Fanuc KAREL source: kt00525.KL

-- PROVISIONAL review KL for V940-1; original PC SHA256 8b3a5a5ea8582134b2ffe9444f4f372b90cdeef2257a1a4dd15e0ae4e4d82a8f
-- Incomplete behavior may be omitted. Consult companion uncertainty JSON. Do not deploy.
PROGRAM KT00525
%NOLOCKGROUP
-- UNRESOLVED_DECL P1 type=000106
-- UNRESOLVED_DECL P2 type=000106
-- UNRESOLVED_DECL OUT type=000102
BEGIN
  -- V9_ZERO_TABLE_METADATA_HINT layout=0001; no indexed target words; source/name/runtime held
  -- UNRESOLVED_PC offsets 5-20; opcodes 2E,22,32,35
  -- UNRESOLVED_PC offsets 25-40; opcodes 2E,22,32,35
  -- UNRESOLVED_PC offsets 45-60; opcodes 2E,22,32,35
  -- UNRESOLVED_PC offsets 65-80; opcodes 2E,22,32,35
  -- UNRESOLVED_PC offsets 85-124; opcodes 49,7E,49,7E,60,7E,4A
  -- UNRESOLVED_PC offsets 129-133; opcodes 7F
END KT00525
